{attribute 'GeneratedUsingTerminal: EL6001-0000-0020'}
{attribute addProperty BoxType "EL6001-0000-0020"}
{attribute addProperty Id "EtcSlaveTerminalBaseCOM_ext_inputsAT %I*COM_ext_inputs_1F197B20108COM_ext_outputsAT %Q*COM_ext_outputs_54D54ACC105WcStateAT %I*WcState_9091E0EB2InfoDataAT %I*InfoData_32EB74EA10"}
{attribute addProperty CRC "592660050"}
{attribute addProperty Size "225"}
TYPE EL6001_23534652 EXTENDS EtcSlaveTerminalBase :
STRUCT
	{attribute addProperty Name "COM_ext_inputs"}
	COM_ext_inputs : COM_ext_inputs_1F197B20;
	{attribute addProperty Name "COM_ext_outputs"}
	COM_ext_outputs : COM_ext_outputs_54D54ACC;
	{attribute addProperty Name "WcState"}
	WcState : WcState_9091E0EB;
	{attribute addProperty Name "InfoData"}
	InfoData : InfoData_32EB74EA;
END_STRUCT
END_TYPE

(* stored: Version 1.2.0.0, ProductVersion 3.1.4024.9
   DUT EL6001_23534652: Id {ab40e735-ae25-47e8-9a3a-8b301c8eb61f} *)
